FUNCTION alg_a_pusher1 : BOOL
VAR_INPUT
	state: STATE;
END_VAR

alg_a_pusher1 := state.dvar_M_inventory1_a_pusher1;

END_FUNCTION

(* stored: Version 1.1.0.1, ProductVersion 3.1.4022.18
   POU alg_a_pusher1: Id {359933f6-17e4-4728-9c0f-90da7cfca5ad}, SpecialFunc None *)
